// TIA Portal V16 export
// export: Created 2024-05-10T06:46:42.5139506Z, ExportSetting WithDefaults, DisplayName Totally Integrated Automation Portal, DisplayVersion V16, DisplayName TIA Portal Version Control Interface, DisplayVersion V16, DisplayName TIA Portal Openness, DisplayVersion V16, DisplayName STEP 7 Professional, DisplayVersion V16, DisplayName STEP 7 Safety, DisplayVersion V16, DisplayName WinCC Professional, DisplayVersion V16
FUNCTION_BLOCK "K22_ST10上自动"   // FB22, LAD
{ S7_Optimized_Access := 'TRUE' }
VERSION : 0.1
// stored: AutoNumber false, IsIECCheckEnabled false, IsRetainMemResEnabled false, MemoryReserve 100, SetENOAutomatically false, UDAEnableTagReadback false
   VAR_TEMP   // added for the SCL form of the ladder/FBD networks
      _w1 : Bool;
   END_VAR
BEGIN

REGION Network 2: @搬出条件，SN12===ST10上工位
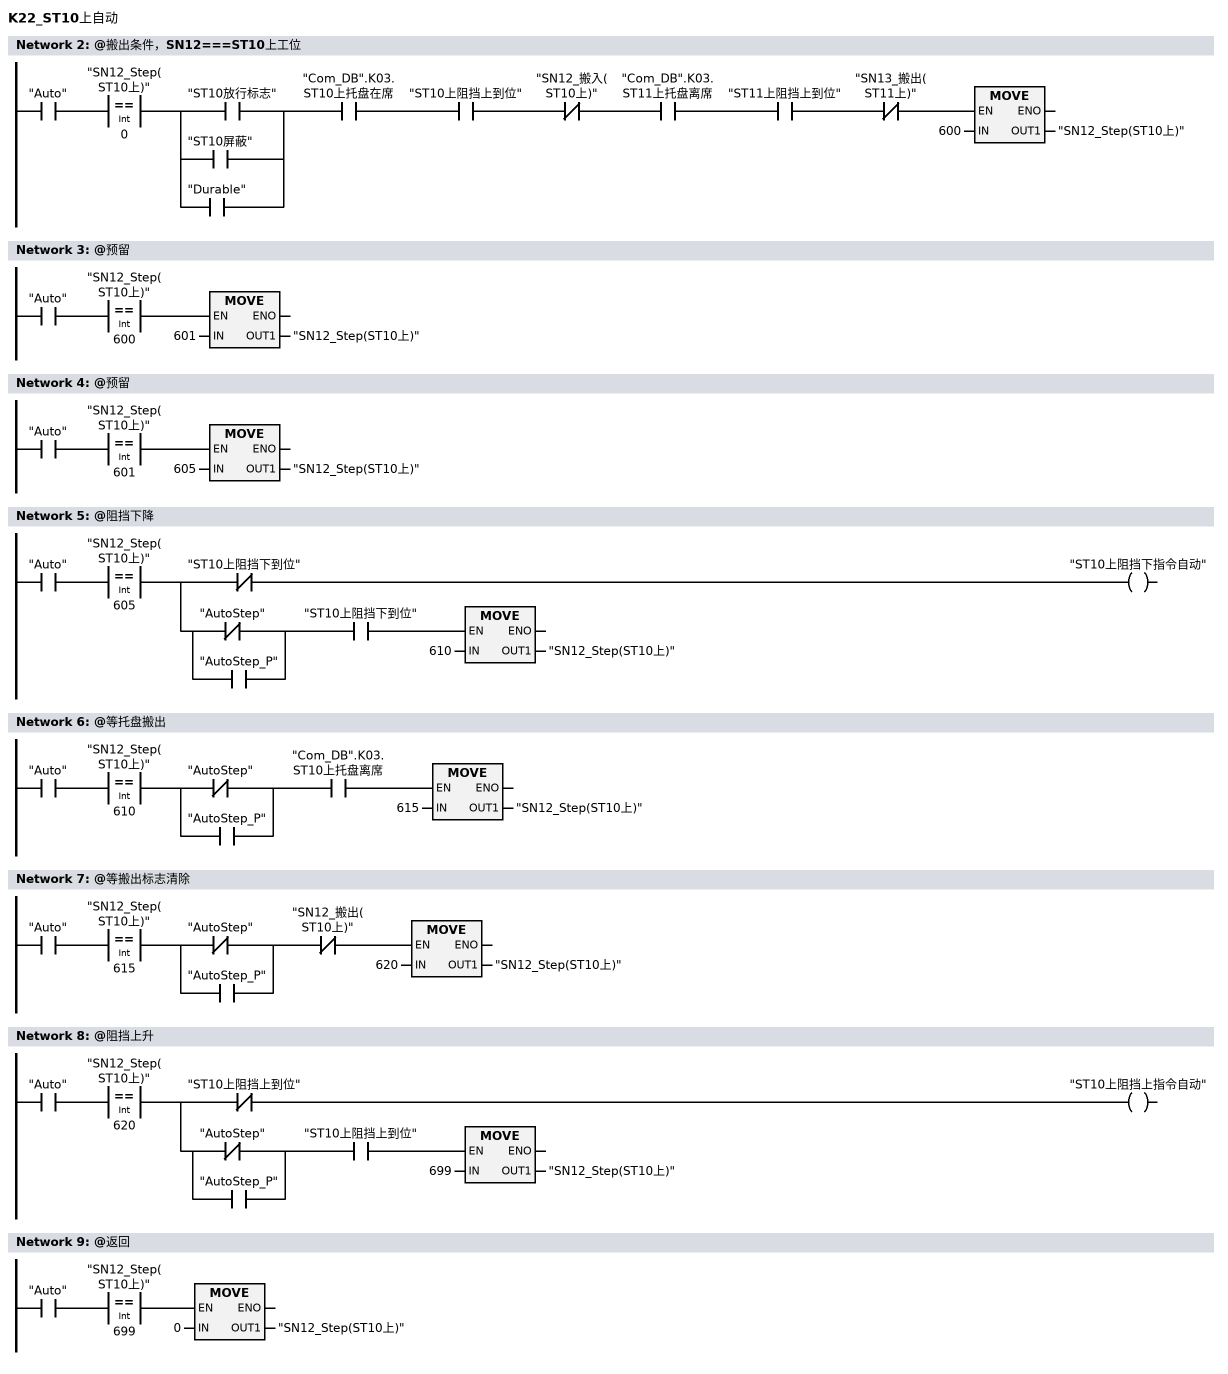
   RUNG wire#powerrail
      Contact( "Auto" )
      { S7_Templates := "SrcType := Int" } EQ_Contact(in1 := "SN12_Step(ST10上)", in2 := 0)
      wire#w1
      Contact( "ST10放行标志" )
      wire#w2
      Contact( "Com_DB".K03.ST10上托盘在席 )
      Contact( "ST10上阻挡上到位" )
      I_Contact( "SN12_搬入(ST10上)" )
      Contact( "Com_DB".K03.ST11上托盘离席 )
      Contact( "ST11上阻挡上到位" )
      I_Contact( "SN13_搬出(ST11上)" )
      Move(in := 600, out1 => "SN12_Step(ST10上)")
   END_RUNG
   RUNG wire#w1
      Contact( "ST10屏蔽" )
   END_RUNG wire#w2
   RUNG wire#w1
      Contact( "Durable" )
   END_RUNG wire#w2
   // the same network as SCL:
   IF "Auto" AND ("SN12_Step(ST10上)" = 0) AND ("ST10放行标志" OR "ST10屏蔽" OR "Durable") AND "Com_DB".K03.ST10上托盘在席 AND "ST10上阻挡上到位" AND NOT "SN12_搬入(ST10上)" AND "Com_DB".K03.ST11上托盘离席 AND "ST11上阻挡上到位" AND NOT "SN13_搬出(ST11上)" THEN
       "SN12_Step(ST10上)" := 600;
   END_IF;
END_REGION

REGION Network 3: @预留
   RUNG wire#powerrail
      Contact( "Auto" )
      { S7_Templates := "SrcType := Int" } EQ_Contact(in1 := "SN12_Step(ST10上)", in2 := 600)
      Move(in := 601, out1 => "SN12_Step(ST10上)")
   END_RUNG
   // the same network as SCL:
   IF "Auto" AND ("SN12_Step(ST10上)" = 600) THEN "SN12_Step(ST10上)" := 601; END_IF;
END_REGION

REGION Network 4: @预留
   RUNG wire#powerrail
      Contact( "Auto" )
      { S7_Templates := "SrcType := Int" } EQ_Contact(in1 := "SN12_Step(ST10上)", in2 := 601)
      Move(in := 605, out1 => "SN12_Step(ST10上)")
   END_RUNG
   // the same network as SCL:
   IF "Auto" AND ("SN12_Step(ST10上)" = 601) THEN "SN12_Step(ST10上)" := 605; END_IF;
END_REGION

REGION Network 5: @阻挡下降
   RUNG wire#powerrail
      Contact( "Auto" )
      { S7_Templates := "SrcType := Int" } EQ_Contact(in1 := "SN12_Step(ST10上)", in2 := 605)
      wire#w1
      I_Contact( "ST10上阻挡下到位" )
      Coil( "ST10上阻挡下指令自动" )
   END_RUNG
   RUNG wire#w1
      I_Contact( "AutoStep" )
      wire#w2
      Contact( "ST10上阻挡下到位" )
      Move(in := 610, out1 => "SN12_Step(ST10上)")
   END_RUNG
   RUNG wire#w1
      Contact( "AutoStep_P" )
   END_RUNG wire#w2
   // the same network as SCL:
   #_w1 := "Auto" AND ("SN12_Step(ST10上)" = 605);
   "ST10上阻挡下指令自动" := #_w1 AND NOT "ST10上阻挡下到位";
   IF #_w1 AND (NOT "AutoStep" OR "AutoStep_P") AND "ST10上阻挡下到位" THEN "SN12_Step(ST10上)" := 610; END_IF;
END_REGION

REGION Network 6: @等托盘搬出
   RUNG wire#powerrail
      Contact( "Auto" )
      { S7_Templates := "SrcType := Int" } EQ_Contact(in1 := "SN12_Step(ST10上)", in2 := 610)
      wire#w1
      I_Contact( "AutoStep" )
      wire#w2
      Contact( "Com_DB".K03.ST10上托盘离席 )
      Move(in := 615, out1 => "SN12_Step(ST10上)")
   END_RUNG
   RUNG wire#w1
      Contact( "AutoStep_P" )
   END_RUNG wire#w2
   // the same network as SCL:
   IF "Auto" AND ("SN12_Step(ST10上)" = 610) AND (NOT "AutoStep" OR "AutoStep_P") AND "Com_DB".K03.ST10上托盘离席 THEN
       "SN12_Step(ST10上)" := 615;
   END_IF;
END_REGION

REGION Network 7: @等搬出标志清除
   RUNG wire#powerrail
      Contact( "Auto" )
      { S7_Templates := "SrcType := Int" } EQ_Contact(in1 := "SN12_Step(ST10上)", in2 := 615)
      wire#w1
      I_Contact( "AutoStep" )
      wire#w2
      I_Contact( "SN12_搬出(ST10上)" )
      Move(in := 620, out1 => "SN12_Step(ST10上)")
   END_RUNG
   RUNG wire#w1
      Contact( "AutoStep_P" )
   END_RUNG wire#w2
   // the same network as SCL:
   IF "Auto" AND ("SN12_Step(ST10上)" = 615) AND (NOT "AutoStep" OR "AutoStep_P") AND NOT "SN12_搬出(ST10上)" THEN
       "SN12_Step(ST10上)" := 620;
   END_IF;
END_REGION

REGION Network 8: @阻挡上升
   RUNG wire#powerrail
      Contact( "Auto" )
      { S7_Templates := "SrcType := Int" } EQ_Contact(in1 := "SN12_Step(ST10上)", in2 := 620)
      wire#w1
      I_Contact( "ST10上阻挡上到位" )
      Coil( "ST10上阻挡上指令自动" )
   END_RUNG
   RUNG wire#w1
      I_Contact( "AutoStep" )
      wire#w2
      Contact( "ST10上阻挡上到位" )
      Move(in := 699, out1 => "SN12_Step(ST10上)")
   END_RUNG
   RUNG wire#w1
      Contact( "AutoStep_P" )
   END_RUNG wire#w2
   // the same network as SCL:
   #_w1 := "Auto" AND ("SN12_Step(ST10上)" = 620);
   "ST10上阻挡上指令自动" := #_w1 AND NOT "ST10上阻挡上到位";
   IF #_w1 AND (NOT "AutoStep" OR "AutoStep_P") AND "ST10上阻挡上到位" THEN "SN12_Step(ST10上)" := 699; END_IF;
END_REGION

REGION Network 9: @返回
   RUNG wire#powerrail
      Contact( "Auto" )
      { S7_Templates := "SrcType := Int" } EQ_Contact(in1 := "SN12_Step(ST10上)", in2 := 699)
      Move(in := 0, out1 => "SN12_Step(ST10上)")
   END_RUNG
   // the same network as SCL:
   IF "Auto" AND ("SN12_Step(ST10上)" = 699) THEN "SN12_Step(ST10上)" := 0; END_IF;
END_REGION
END_FUNCTION_BLOCK
